INTERFACE I_Sequenz

METHOD M_Start : BOOL
VAR_INPUT
END_VAR
END_METHOD

METHOD M_Stop : BOOL
VAR_INPUT
END_VAR
END_METHOD

PROPERTY P_Finished : BOOL;
GET
END_GET
END_PROPERTY

END_INTERFACE

(* stored: Version 1.1.0.1
   Itf I_Sequenz: Id {28ceae57-4089-44a8-ae28-9022f28b8d95}
   Method M_Start: Id {7595f5ae-7473-40a2-b38e-71430a151be1}
   Method M_Stop: Id {3ff0a064-1a84-478c-95ab-766dafd5e58d}
   Property P_Finished: Id {3b9ebe4a-5c53-4138-8556-733b227a563a}
   Get Get: Id {f368a448-4439-40c5-9e56-558186d7d188} *)
